GLOBALCONSTANTS ISOUSERHOME_e (* CF / User network location *)
  (* Standard: 61499-1 *)
  (* Version 1.0, 2025-10-18, Franz Höpfinger *)
  PACKAGE isobus::pgn;
  VAR_GLOBAL CONSTANT
    intern : SINT := 0;
    network : SINT := 1; (* < Internal CF / user *)
    thisMember : SINT := 2; (* < External CF / user *)
    notdef : SINT := -1; (* < Event is for this internal CF / user *)
  END_VAR
END_GLOBALCONSTANTS
